(* Schneider Machine Expert - Basic project sequential_lights_TM221CE40T, file version 3.0.0.0 *)
(* ProjectInformations: Name=Sequential Lights TM221CE40T *)

HARDWARE
  Cpu 0: TM221CE40T
  EthernetConfiguration: NetworkName=M221, IpAllocationMode=ByDhcp, IpAddress=192.168.1.10, SubnetMask=255.255.255.0
  SerialLineConfiguration: Baud=Baud19200, Parity=ParityEven, DataBits=DataBits8, StopBits=StopBits1, PhysicalMedium=PhysicalMediumRs485, TransmissionMode=TransmissionModeModbusRtu, SlaveId=1, Addressing=SlaveAddressing
  MastTask: UsePeriodScanMode=false, PeriodScan=100
  FastTask: Period=255
  CpuBehavior: StartingMode=StartAsPreviousState, AutoSaveRamOnEeprom=true, WatchdogPeriod=250

SYMBOLS  (address, symbol, comment, settings)
  %M0       AUTO_RUN  "Auto sequence running flag"
  %M1       TMR0_DONE  "Timer 0 done flag"
  %M2       TMR1_DONE  "Timer 1 done flag"
  %TM0        [Preset=5, Base=OneSecond]
  %TM1        [Preset=5, Base=OneSecond]
  %I0.0     MODE_AUTO
  %I0.1     PB_START
  %I0.2     ESTOP
  %I0.3     LIGHT1_SW
  %I0.4     LIGHT2_SW
  %I0.5     LIGHT3_SW
  %Q0.0     LIGHT1
  %Q0.1     LIGHT2
  %Q0.2     LIGHT3

POU Sequential Lights Control
  (* SectionNumber=1 *)

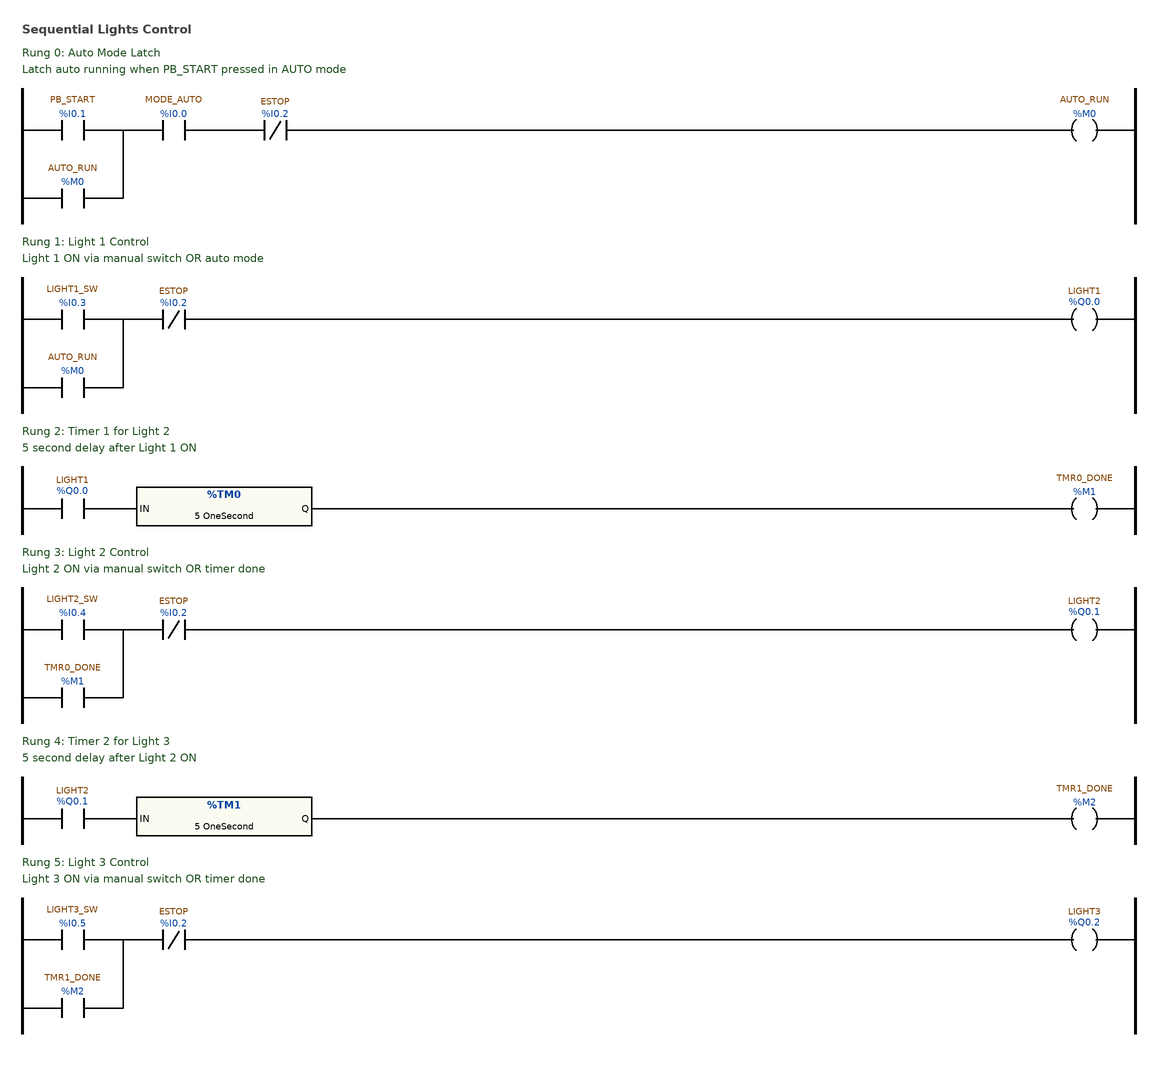

// Rung 0: Auto Mode Latch
// Latch auto running when PB_START pressed in AUTO mode
  LD %I0.1                (* PB_START *)
  OR %M0                  (* AUTO_RUN *)
  AND %I0.0               (* MODE_AUTO *)
  ANDN %I0.2              (* ESTOP *)
  ST %M0                  (* AUTO_RUN *)
  // as ST:
  //   AUTO_RUN := (PB_START OR AUTO_RUN) AND MODE_AUTO AND NOT ESTOP;

// Rung 1: Light 1 Control
// Light 1 ON via manual switch OR auto mode
  LD %I0.3                (* LIGHT1_SW *)
  OR %M0                  (* AUTO_RUN *)
  ANDN %I0.2              (* ESTOP *)
  ST %Q0.0                (* LIGHT1 *)
  // as ST:
  //   LIGHT1 := (LIGHT1_SW OR AUTO_RUN) AND NOT ESTOP;

// Rung 2: Timer 1 for Light 2
// 5 second delay after Light 1 ON
  BLK %TM0
  LD %Q0.0                (* LIGHT1 *)
  IN
  OUT_BLK
  LD Q
  ST %M1                  (* TMR0_DONE *)
  END_BLK
  // as ST:
  //   %TM0(IN := LIGHT1);
  //   TMR0_DONE := %TM0.Q;

// Rung 3: Light 2 Control
// Light 2 ON via manual switch OR timer done
  LD %I0.4                (* LIGHT2_SW *)
  OR %M1                  (* TMR0_DONE *)
  ANDN %I0.2              (* ESTOP *)
  ST %Q0.1                (* LIGHT2 *)
  // as ST:
  //   LIGHT2 := (LIGHT2_SW OR TMR0_DONE) AND NOT ESTOP;

// Rung 4: Timer 2 for Light 3
// 5 second delay after Light 2 ON
  BLK %TM1
  LD %Q0.1                (* LIGHT2 *)
  IN
  OUT_BLK
  LD Q
  ST %M2                  (* TMR1_DONE *)
  END_BLK
  // as ST:
  //   %TM1(IN := LIGHT2);
  //   TMR1_DONE := %TM1.Q;

// Rung 5: Light 3 Control
// Light 3 ON via manual switch OR timer done
  LD %I0.5                (* LIGHT3_SW *)
  OR %M2                  (* TMR1_DONE *)
  ANDN %I0.2              (* ESTOP *)
  ST %Q0.2                (* LIGHT3 *)
  // as ST:
  //   LIGHT3 := (LIGHT3_SW OR TMR1_DONE) AND NOT ESTOP;
